// TIA Portal V18 export
// export: Created 2026-01-09T11:23:37.0161229Z, ExportSetting WithDefaults, DisplayName Totally Integrated Automation Portal, DisplayVersion V18 Update 5, DisplayName TIA Portal Openness, DisplayVersion V18 Update 5, DisplayName TIA Portal Teamcenter Gateway, DisplayVersion V18, DisplayName TIA Portal Version Control Interface, DisplayVersion V18, DisplayName SINAMICS Startdrive Advanced, DisplayVersion V18 SP2 Update 1, DisplayName SINAMICS Startdrive G110M, G120, G120C, G120D, G120P, G115D, DisplayVersion V18 SP2 Update 1, DisplayName SINAMICS Startdrive G130, G150, S120, S150, SINAMICS MV, S210, G220, S200, DisplayVersion V18 SP2 Update 1, DisplayName STEP 7 Professional, DisplayVersion V18 Update 5, DisplayName STEP 7 Safety, DisplayVersion V18, DisplayName WinCC Professional, DisplayVersion V18 Update 5
Screen "290_Cylinder_L1"  1280x800, Number=290, Template=02ManualUnit1
  ScreenLayer "Layer_0"
    FaceplateInstance "Cylinder_S71500_TP700_1" at 0,85 size 1279x80  FaceplateTypeName=03 FunctionBlocks@$@101 Cylinder@$@101.2 HMI@$@S7-1500@$@Cylinder_S71500_TP700 V 0.0.29
      Cy := STxxxCylinder051
      CylinderName := Cyl name
      HomeButtonName := Cyl go home button
      WorkButtonName := Cyl go work button
      HomeQaddress := Cyl home Q
      HomeIaddress := Cyl home I
      WorkIaddress := Cyl work I
      WorkQaddress := Cyl work Q
    FaceplateInstance "Cylinder_S71500_TP700_3" at 0,160 size 1279x80  FaceplateTypeName=03 FunctionBlocks@$@101 Cylinder@$@101.2 HMI@$@S7-1500@$@Cylinder_S71500_TP700 V 0.0.29
      Cy := STxxxCylinder052
      CylinderName := Cyl name
      HomeButtonName := Cyl go home button
      WorkButtonName := Cyl go work button
      HomeQaddress := Cyl home Q
      HomeIaddress := Cyl home I
      WorkIaddress := Cyl work I
      WorkQaddress := Cyl work Q
    Button "btnMenu6" at 640,725 size 128x75  Mode=Text, StyleItem=BtnNormal20
    Button "btnMenu6_1" at 768,725 size 128x75  Mode=Text, StyleItem=BtnNormal20
    Button "btnMenu4" at 384,725 size 128x75  Mode=Text, TextOff="L-气缸2 / L-Cylinder2", TextOn="L-气缸2 / L-Cylinder2"
      on Click: ActivateScreen(Screen name := 293_Cylinder_L2, Object number := 0)
    Button "btnMenu5" at 512,725 size 128x75  Mode=Text, TextOff="L-电机2 / L-Motor2", TextOn="L-电机2 / L-Motor2"
      on Click: ActivateScreen(Screen name := 294_Motor_L2, Object number := 0)
    Button "btnMenu7" at 896,725 size 128x75  Mode=Text
    Button "btnMenu7_1" at 1024,725 size 128x75  Mode=Text
    Button "按钮_9" at 128,725 size 128x75  Mode=Text, PictureOff=向右箭头_0, TextOff="L-气缸1 / L-Cylinder1", TextOn="L-气缸1 / L-Cylinder1"
      on Click: ActivateScreen(Screen name := , Object number := 0)
    Button "btnMenu4_1" at 256,725 size 128x75  Mode=Text, TextOff="L-电机1 / L-Motor1", TextOn="L-电机1 / L-Motor1"
      on Click: ActivateScreen(Screen name := 291_Motor_L1, Object number := 0)
    GraphicView "图形视图_1" at 45,248 size 1194x412  Picture=图形_60
